(* IEC 61131-3 sources: Lasal/CPU_5344_V01/Class/gbl_datatypes, 1 file *)

(* ---- gbl_datatypes.st ---- *)
(*!
<Class
	Name               = "gbl_datatypes"
	Revision           = "0.0"
	RealtimeTask       = "false"
	CyclicTask         = "false"
	BackgroundTask     = "false"
	Sigmatek           = "false"
	OSInterface        = "false"
	HighPriority       = "false"
	Automatic          = "false"
	UpdateMode         = "Prescan"
	SharedCommandTable = "true"
	Objectsize         = "(284,120)">
	<Channels>
		<Server Name="ClassSvr" Visualized="false" Initialize="false" WriteProtected="true" Retentive="false"/>
	</Channels>
</Class>
*)
gbl_datatypes : CLASS
	TYPE
	  tStr13 : ARRAY [0..12] OF CHAR;  //! <Type Public="true" Name="tStr13"/>
	  tStr20 : ARRAY [0..19] OF CHAR;  //! <Type Public="true" Name="tStr20"/>
	  tStr25 : ARRAY [0..24] OF CHAR;  //! <Type Public="true" Name="tStr25"/>
	END_TYPE
  //Servers:
	ClassSvr 	: SvrChCmd_DINT;
  //Clients:
  //Variables:
  //Functions:
  //Tables:
	FUNCTION @STD
		VAR_OUTPUT
			ret_code	: CONFSTATES;
		END_VAR;
	FUNCTION GLOBAL TAB @CT_;
END_CLASS;
